// TIA Portal V20 export
DATA_BLOCK "Data"   // DB40
// stored: Access Published, MemoryReserve 100, Namespace Global
   VAR
      general : "LAF_typeGeneralStatus";   // Global status information
      unit : Array[0.._.NO_OF_UNITS] of "LAF_typeUnitInterface";   // Global information of units
   END_VAR
BEGIN
   // general.enablePower : Power is off. Switch on!
   unit[0].enableControlInterfaces.local := TRUE;
   unit[0].enableControlInterfaces.hmi := FALSE;
   // unit[0].specialFunctions.HoursTest : FAT_Hours Test
   // unit[0].specialFunctions.Capability : FAT_Capability
   // unit[0].specialFunctions.Sampling : FAT_Sampling
END_DATA_BLOCK
